// Mitsubishi GX Works2 project: 0709flt int   PLC: Q02/Q02H

PROGRAM MAIN
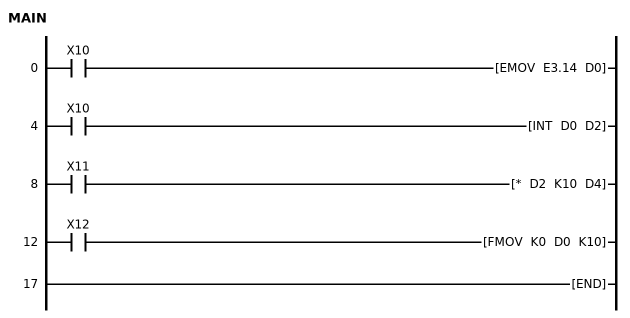
0     LD      X10
      EMOV    E3.14 D0
4     LD      X10
      INT     D0 D2
8     LD      X11
      *       D2 K10 D4
12    LD      X12
      FMOV    K0 D0 K10
17    END
END_PROGRAM
